{attribute 'pack_mode' := '0'}
TYPE ACMethodMixingP EXTENDS ACMethodBaseP : 
STRUCT
	// Ausschalten 
	_SwitchOff : BOOL;
	// Geschwindigkeit 
	_Speed : INT;
	// Mindestgewicht 
	_MinWeight : LREAL;
	// Dauer 
	_Duration : TIME;
	// Temperatur 
	_Temperature : LREAL;
	
END_STRUCT
END_TYPE

(* stored: Version 1.1.0.1, ProductVersion 3.1.4020.12
   DUT ACMethodMixingP: Id {a2a6c75c-c379-49f3-9a67-2efd8c51483a} *)
